// TIA Portal project "Data Logging" (V11)

(* hardware
DEVICE "SIMATIC 1200 station_1"  S71200.Device
   slot 0: "S7-1200 rack"  Rack  V1.0
   slot 1: "S71200-1001203"  CPU 1214C DC/DC/DC  6ES7 214-1AE30-0XB0  V2.0
*)

// ===== PLC "S71200-1001203"  CPU 1214C DC/DC/DC =====

VAR_GLOBAL   // PLC tag table "Default tag table"
   "System_Byte" AT %MB1 : Byte;
   "FirstScan" AT %M1.0 : Bool;
   "DiagStatusUpdate" AT %M1.1 : Bool;
   "AlwaysTRUE" AT %M1.2 : Bool;
   "AlwaysFALSE" AT %M1.3 : Bool;
   "Clock_Byte" AT %MB0 : Byte;
   "Clock_10Hz" AT %M0.0 : Bool;
   "Clock_5Hz" AT %M0.1 : Bool;
   "Clock_2.5Hz" AT %M0.2 : Bool;
   "Clock_2Hz" AT %M0.3 : Bool;
   "Clock_1.25Hz" AT %M0.4 : Bool;
   "Clock_1Hz" AT %M0.5 : Bool;
   "Clock_0.625Hz" AT %M0.6 : Bool;
   "Clock_0.5Hz" AT %M0.7 : Bool;
   "Last Create Error Status" AT %MW2 : Word;
   "auxp1" AT %M4.0 : Bool;
   "Nr create Ok" AT %MW6 : Int;
   "auxp2" AT %M4.1 : Bool;
   "Nr create error" AT %MW8 : Int;
   "Command Create" AT %M4.2 : Bool;
   "Command Write" AT %M4.3 : Bool;
   "Last Write Error Status" AT %MW10 : Word;
   "auxp3" AT %M4.4 : Bool;
   "Nr Write Ok" AT %MW12 : Int;
   "auxp4" AT %M4.5 : Bool;
   "Nr Write error" AT %MW14 : Int;
   "Nr Open Error" AT %MW16 : Int;
   "Nr Open Dones" AT %MW18 : Int;
   "Last Open Error Status" AT %MW20 : Word;
   "Nr Close Error" AT %MW22 : Int;
   "Nr Close Done" AT %MW24 : Int;
   "Last Close Error Status" AT %MW26 : Word;
   "Nr New Error" AT %MW28 : Int;
   "Nr New Dones" AT %MW30 : Int;
   "Last New Status" AT %MW32 : Word;
   "Command Open" AT %M4.6 : Bool;
   "Command Close" AT %M4.7 : Bool;
   "command New" AT %M5.0 : Bool;
   "Open Mode" AT %MW36 : UInt;
   "Nr_records" AT %MW34 : UInt;
END_VAR

DATA_BLOCK "Data_block_1"   // DB2
{ S7_Optimized_Access := 'FALSE' }
VERSION : 0.1
   VAR
      "Archiev Name" : String := 'Banana';
      ID : DWord;
      Header : String := ' Var1, Var2';
      Data : Struct
         Int1 : Int;
         real1 : Real;
      END_STRUCT;
   END_VAR
BEGIN
END_DATA_BLOCK

DATA_BLOCK "Diag Create"   // DB5
{ S7_Optimized_Access := 'FALSE' }
VERSION : 0.1
// stored: InstanceOfName Block_Diag
"Block_Diag"
BEGIN
END_DATA_BLOCK

DATA_BLOCK "Diag Write"   // DB6
{ S7_Optimized_Access := 'FALSE' }
VERSION : 0.1
// stored: InstanceOfName Block_Diag
"Block_Diag"
BEGIN
END_DATA_BLOCK

DATA_BLOCK "Diag Open"   // DB7
{ S7_Optimized_Access := 'FALSE' }
VERSION : 0.1
// stored: InstanceOfName Block_Diag
"Block_Diag"
BEGIN
END_DATA_BLOCK

DATA_BLOCK "Diag Close"   // DB10
{ S7_Optimized_Access := 'FALSE' }
VERSION : 0.1
// stored: InstanceOfName Block_Diag
"Block_Diag"
BEGIN
END_DATA_BLOCK

DATA_BLOCK "Diag New File"   // DB11
{ S7_Optimized_Access := 'FALSE' }
VERSION : 0.1
// stored: InstanceOfName Block_Diag
"Block_Diag"
BEGIN
END_DATA_BLOCK

FUNCTION_BLOCK "Block_Diag"   // FB1, LAD
{ S7_Optimized_Access := 'FALSE' }
VERSION : 0.1
   VAR_INPUT
      Error : Bool;
      Done : Bool;
      Status : Word;
   END_VAR
   VAR_OUTPUT
      Nr_Errors : Int;
      Nr_Dones : Int;
      Last_Status : Word;
   END_VAR
   VAR
      P1 : Bool;
      P2 : Bool;
   END_VAR
   VAR_TEMP   // added for the SCL form of the ladder/FBD networks
      _w1 : Bool;
   END_VAR
BEGIN

REGION Network 1
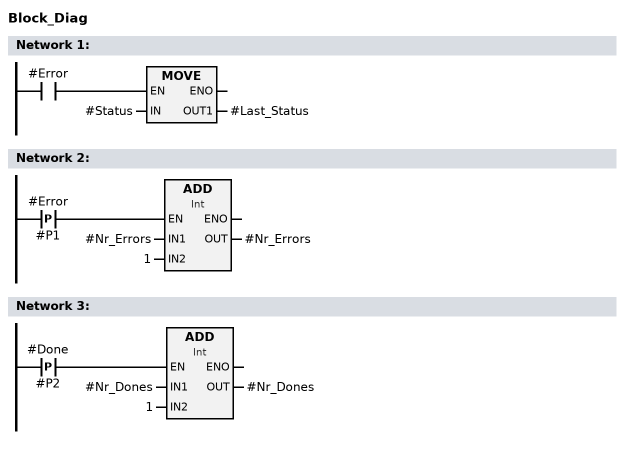
   RUNG wire#powerrail
      Contact( #Error )
      { S7_GenerateENO := "TRUE" } Move(in := #Status, out1 => #Last_Status)
   END_RUNG
   // the same network as SCL:
   IF #Error THEN #Last_Status := #Status; END_IF;
END_REGION

REGION Network 2
   RUNG wire#powerrail
      P_Contact(operand := #Error, bit := #P1)
      { S7_Templates := "SrcType := Int"; S7_GenerateENO := "TRUE" } Add(in1 := #Nr_Errors, in2 := 1, out => #Nr_Errors)
   END_RUNG
   // the same network as SCL:
   #_w1 := #Error AND NOT #P1;   // rising edge of #Error
   #P1 := #Error;
   IF #_w1 THEN #Nr_Errors := #Nr_Errors + 1; END_IF;
END_REGION

REGION Network 3
   RUNG wire#powerrail
      P_Contact(operand := #Done, bit := #P2)
      { S7_Templates := "SrcType := Int"; S7_GenerateENO := "TRUE" } Add(in1 := #Nr_Dones, in2 := 1, out => #Nr_Dones)
   END_RUNG
   // the same network as SCL:
   #_w1 := #Done AND NOT #P2;   // rising edge of #Done
   #P2 := #Done;
   IF #_w1 THEN #Nr_Dones := #Nr_Dones + 1; END_IF;
END_REGION
END_FUNCTION_BLOCK

ORGANIZATION_BLOCK "Main"   // OB1, LAD, ProgramCycle
TITLE = "Main Program Sweep (Cycle)"
{ S7_Optimized_Access := 'FALSE' }
VERSION : 0.1
BEGIN
END_ORGANIZATION_BLOCK